Universal Robots PolyScope program: Programa_iniciales.urp

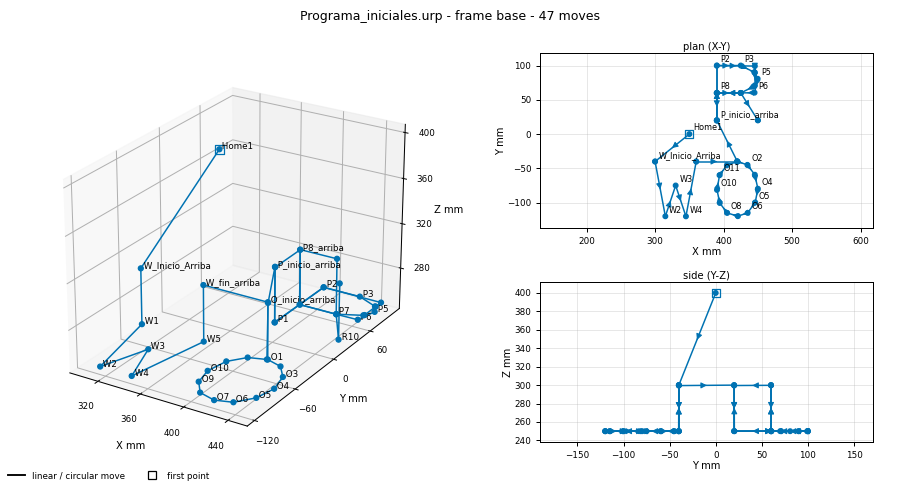
[picture p0: tool path of Programa_iniciales.urp in frame base, 47 of 47 moves have a stored position in this frame; points joined in program order, loops and branches not executed]
Program Programa_iniciales (installation=lab_manipulador directory=/ursim/programs createdIn=3.15.8.106339 lastSavedIn=3.15.8.106339 robotSerialNumber=2018359999)
Calibrated DH parameters: a=[0, -0.425, -0.39225, 0, 0, 0]; d=[0.089159, 0, 0, 0.10915, 0.09465, 0.0823]; alpha=[1.570796, 0, 0, 1.570796, -1.570796, 0]; deltaTheta=[0, 0, 0, 0, 0, 0]
Robot Program (runOnlyOnce=true)
  MoveJ speed 60 deg/s, acceleration 80 deg/s^2 (useActiveTCP=true)
    Waypoint Home1: TCP in base x=350 y=0 z=400 mm, rx=0 ry=3.1412 rz=0 rad; joints [18.173, -68.7, -111.718, -89.559, 89.993, 108.173] deg
    Popup Message (haltProgram=false message=Se simulara la letra W del integrante con iniciales WO inputType=Text)
    MoveL speed 50 mm/s, acceleration 100 mm/s^2 (useActiveTCP=true) feature=Base
      Waypoint W_Inicio_Arriba: TCP in base x=300 y=-40 z=300 mm, rx=0 ry=3.1412 rz=0 rad; joints [13.547, -62.614, -129.791, -77.572, 89.995, 103.547] deg
      Waypoint W1: TCP in base x=300 y=-40 z=250 mm, rx=0 ry=-3.1412 rz=0 rad; joints [13.543, -65.298, -136.072, -68.653, 90.005, 103.543] deg
      Waypoint W2: TCP in base x=314.979 y=-119.886 z=250 mm, rx=0 ry=-3.1412 rz=0 rad; joints [-1.941, -71.65, -132.457, -65.917, 89.999, 88.059] deg
      Waypoint W3: TCP in base x=330 y=-75.001 z=250 mm, rx=0 ry=-3.1412 rz=0 rad; joints [6.011, -71.895, -132.303, -65.825, 90.002, 96.011] deg
      Waypoint W4: TCP in base x=345 y=-120 z=250 mm, rx=0 ry=-3.1412 rz=0 rad; joints [-1.792, -76.456, -129.227, -64.34, 89.999, 88.208] deg
      Waypoint W5: TCP in base x=359.987 y=-40.067 z=250 mm, rx=0 ry=-3.1412 rz=0 rad; joints [11.186, -75.952, -129.588, -64.484, 90.005, 101.186] deg
      Waypoint W_fin_arriba: TCP in base x=360 y=-40 z=299.962 mm, rx=0 ry=-3.1412 rz=0 rad; joints [11.197, -72.92, -123.84, -73.262, 90.005, 101.197] deg
      Popup Message (haltProgram=false message=Se simuara la letra O del integrante con las iniciales WO inputType=Text)
      Waypoint O_inicio_arriba: TCP in base x=419.789 y=-40 z=300 mm, rx=0 ry=-3.1412 rz=0 rad; joints [9.557, -82.138, -116.881, -71.004, 90.004, 99.557] deg
      Waypoint O1: TCP in base x=420 y=-40 z=250.005 mm, rx=0 ry=-3.1412 rz=0 rad; joints [9.552, -85.22, -122.151, -62.652, 90.004, 99.552] deg
      Waypoint O2: TCP in base x=434.653 y=-44.884 z=250.005 mm, rx=0 ry=-3.1412 rz=0 rad; joints [8.569, -87.397, -120.145, -62.481, 90.003, 98.569] deg
      Waypoint O3: TCP in base x=445.447 y=-59.263 z=250.005 mm, rx=0 ry=-3.1412 rz=0 rad; joints [6.479, -89.152, -118.455, -62.416, 90.003, 96.479] deg
      Waypoint O4: TCP in base x=449.93 y=-79.683 z=250.005 mm, rx=0 ry=-3.1412 rz=0 rad; joints [3.777, -90.205, -117.409, -62.409, 90.002, 93.777] deg
      Waypoint O5: TCP in base x=446.074 y=-99.619 z=250.005 mm, rx=0 ry=-3.1412 rz=0 rad; joints [1.227, -90.223, -117.391, -62.409, 90.001, 91.227] deg
      Waypoint O6: TCP in base x=435.084 y=-114.883 z=250.005 mm, rx=0 ry=-3.1412 rz=0 rad; joints [-0.754, -89.239, -118.369, -62.415, 90, 89.246] deg
      Waypoint O7: TCP in base x=420.801 y=-119.728 z=250.005 mm, rx=0 ry=-3.1412 rz=0 rad; joints [-1.435, -87.474, -120.073, -62.477, 89.999, 88.565] deg
      Waypoint O8: TCP in base x=405.118 y=-115.035 z=250 mm, rx=0 ry=-3.1412 rz=0 rad; joints [-0.831, -85.108, -122.252, -62.663, 90, 89.169] deg
      Waypoint O9: TCP in base x=394.351 y=-100.475 z=250 mm, rx=0 ry=-3.1412 rz=0 rad; joints [1.264, -83.002, -124.093, -62.929, 90.001, 91.264] deg
      Waypoint O10: TCP in base x=390.301 y=-81.415 z=250 mm, rx=0 ry=-3.1412 rz=0 rad; joints [4.105, -81.751, -125.142, -63.13, 90.002, 94.105] deg
      Waypoint O11: TCP in base x=393.996 y=-60.022 z=250 mm, rx=0 ry=-3.1412 rz=0 rad; joints [7.232, -81.727, -125.162, -63.135, 90.003, 97.232] deg
      Waypoint O12: TCP in base x=404.711 y=-45.394 z=250 mm, rx=0 ry=-3.1412 rz=0 rad; joints [9.146, -83.047, -124.054, -62.922, 90.004, 99.146] deg
      Waypoint O13: TCP in base x=419.344 y=-40.231 z=250 mm, rx=0 ry=-3.1412 rz=0 rad; joints [9.536, -85.128, -122.235, -62.661, 90.004, 99.536] deg
      Waypoint O_fin_arriba: TCP in base x=419.993 y=-40.002 z=299.487 mm, rx=0 ry=-3.1412 rz=0 rad; joints [9.552, -82.194, -116.913, -70.916, 90.004, 99.552] deg
      Popup Message (haltProgram=false message=Se simulara la letra P del integrante con las iniciales PR inputType=Text)
      Waypoint P_inicio_arriba: TCP in base x=390.034 y=19.933 z=299.999 mm, rx=0 ry=-3.1412 rz=0 rad; joints [19.153, -77.422, -120.641, -71.959, 90.008, 109.153] deg
      Waypoint P1: TCP in base x=390 y=20 z=250.142 mm, rx=0 ry=-3.1412 rz=0 rad; joints [19.165, -80.479, -126.153, -63.391, 90.008, 109.165] deg
      Waypoint P2: TCP in base x=390 y=99.857 z=250 mm, rx=0 ry=-3.1412 rz=0 rad; joints [30.09, -82.342, -124.651, -63.027, 90.012, 120.09] deg
      Waypoint P3: TCP in base x=424.921 y=100 z=250 mm, rx=0 ry=-3.1412 rz=0 rad; joints [27.721, -87.336, -120.205, -62.481, 90.011, 117.721] deg
      Waypoint P4: TCP in base x=444.816 y=90.092 z=250.001 mm, rx=0 ry=-3.1412 rz=0 rad; joints [25.364, -89.777, -117.838, -62.406, 90.01, 115.364] deg
      Waypoint P5: TCP in base x=449.622 y=80.737 z=250 mm, rx=0 ry=-3.1412 rz=0 rad; joints [24.002, -90.189, -117.427, -62.406, 90.01, 114.002] deg
      Waypoint P6: TCP in base x=445.096 y=60.428 z=250 mm, rx=0 ry=-3.1412 rz=0 rad; joints [21.793, -89.125, -118.482, -62.414, 90.009, 111.793] deg
      Waypoint P7: TCP in base x=425.028 y=60.001 z=250 mm, rx=0 ry=-3.1412 rz=0 rad; joints [22.765, -86.289, -121.18, -62.553, 90.009, 112.765] deg
      Waypoint P8: TCP in base x=390.001 y=60.001 z=250 mm, rx=0 ry=-3.1412 rz=0 rad; joints [24.802, -81.12, -125.659, -63.242, 90.01, 114.803] deg
      Waypoint P8_arriba: TCP in base x=390.001 y=60.001 z=299.774 mm, rx=0 ry=-3.1412 rz=0 rad; joints [24.802, -78.059, -120.194, -71.769, 90.01, 114.803] deg
      Popup Message (haltProgram=false message=Se simulara la letra R inputType=Text)
      Waypoint R_inicio_arriba: TCP in base x=390.145 y=20 z=299.565 mm, rx=0 ry=-3.1412 rz=0 rad; joints [19.157, -77.461, -120.679, -71.883, 90.008, 109.157] deg
      Waypoint R1: TCP in base x=390.145 y=20 z=250 mm, rx=0 ry=-3.1412 rz=0 rad; joints [19.157, -80.512, -126.15, -63.361, 90.008, 109.157] deg
      Waypoint R2: TCP in base x=390.145 y=99.998 z=250 mm, rx=0 ry=-3.1412 rz=0 rad; joints [30.098, -82.369, -124.628, -63.023, 90.012, 120.098] deg
      Waypoint R3: TCP in base x=445.503 y=99.205 z=250 mm, rx=0 ry=-3.1412 rz=0 rad; joints [26.388, -90.134, -117.482, -62.405, 90.01, 116.388] deg
      Waypoint R4: TCP in base x=445.503 y=89.942 z=250 mm, rx=0 ry=-3.1412 rz=0 rad; joints [25.308, -89.867, -117.749, -62.405, 90.01, 115.308] deg
      Waypoint R5: TCP in base x=445.503 y=71.068 z=250 mm, rx=0 ry=-3.1412 rz=0 rad; joints [23.063, -89.399, -118.213, -62.41, 90.009, 113.063] deg
      Waypoint R6: TCP in base x=444.95 y=69.954 z=250.046 mm, rx=0 ry=-3.1412 rz=0 rad; joints [22.957, -89.295, -118.308, -62.419, 90.009, 112.957] deg
      Waypoint R7: TCP in base x=425.101 y=60.05 z=250.046 mm, rx=0 ry=-3.1412 rz=0 rad; joints [22.767, -86.297, -121.165, -62.56, 90.009, 112.767] deg
      Waypoint R8: TCP in base x=390.454 y=60.05 z=250.046 mm, rx=0 ry=-3.1412 rz=0 rad; joints [24.781, -81.187, -125.597, -63.237, 90.01, 114.781] deg
      Waypoint R8_arriba: TCP in base x=390 y=60 z=299.944 mm, rx=0 ry=-3.1412 rz=0 rad; joints [24.802, -78.05, -120.174, -71.797, 90.01, 114.802] deg
      Popup Message (haltProgram=false message=Se simulara la letra R.Trazo 2:diagonal inputType=Text)
      Waypoint R9_arriba: TCP in base x=424.753 y=60 z=300 mm, rx=0 ry=-3.1412 rz=0 rad; joints [22.779, -83.21, -115.966, -70.846, 90.009, 112.779] deg
      Waypoint R9: TCP in base x=424.999 y=60 z=250.159 mm, rx=0 ry=-3.1412 rz=0 rad; joints [22.766, -86.273, -121.169, -62.58, 90.009, 112.766] deg
      Waypoint R10: TCP in base x=449.851 y=20.239 z=250.001 mm, rx=0 ry=-3.1412 rz=0 rad; joints [16.602, -89.283, -118.327, -62.413, 90.007, 106.602] deg
      Waypoint R_fin_arriba: TCP in base x=450 y=20 z=299.918 mm, rx=0 ry=-3.1412 rz=0 rad; joints [16.567, -86.315, -113.199, -70.509, 90.007, 106.567] deg
